PROGRAM MAIN
VAR
	fb_rcp : FB_RPC;
END_VAR

END_PROGRAM

(* stored: Version 1.1.0.1, ProductVersion 3.1.4024.12
   POU MAIN: Id {b287065f-b8ee-4be1-a1a7-426c57644ca7}, SpecialFunc None *)
